INTERFACE I_XP_Environment  EXTENDS __SYSTEM.IQueryInterface, I_CH_Object

METHOD AddToGroup : HRESULT
VAR_INPUT
	iGroup : I_XP_Group;
END_VAR
END_METHOD

METHOD Clear : HRESULT
END_METHOD

METHOD Configure : HRESULT
VAR_INPUT
END_VAR
END_METHOD

{attribute 'monitoring':='call'}
PROPERTY Feedback : I_XP_Feedback
GET
END_GET
END_PROPERTY

METHOD Initialize : HRESULT
END_METHOD

{attribute 'monitoring':='call'}
PROPERTY Mapped : BOOL //Project is mapped to MC (McToPlc and PlcToMc)
GET
END_GET
END_PROPERTY

{attribute 'monitoring':='call'}
//Unique object ID
PROPERTY OID : OTCID
GET
END_GET
END_PROPERTY

{attribute 'monitoring':='call'}
PROPERTY PlanarEnvironment : REFERENCE TO MC_PlanarEnvironment
GET
END_GET
END_PROPERTY

METHOD RemoveFromGroup : HRESULT
END_METHOD

METHOD PUBLIC Update : HRESULT
VAR_INPUT
END_VAR
END_METHOD

{attribute 'monitoring':='call'}
PROPERTY UtilityEnvirement : Tc3_XPlanarUtility.I_Environment
GET
END_GET
END_PROPERTY

END_INTERFACE

(* stored: Version 1.1.0.1, ProductVersion 3.1.4024.12
   Itf I_XP_Environment: Id {82d4e6a8-d939-49b0-818e-86b258207442}
   Method AddToGroup: Id {f4493e59-ad90-4dac-89cb-3c35b7abff5c}
   Method Clear: Id {2eaf657c-b06a-4ac5-8bfd-2f4b4ad6572c}
   Method Configure: Id {9bbca1e7-a2f1-485d-8de7-8f90a1dc3677}
   Property Feedback: Id {e6ee7906-45bb-443c-afb3-2b2a9b508770}
   Get Get: Id {cc18bd10-41f4-4051-8a16-631b92b39a61}
   Method Initialize: Id {0d86c81e-3fa8-49c7-87ef-1a4588a06d1e}
   Property Mapped: Id {14b61345-b383-42ca-9c63-97777c6507b6}
   Get Get: Id {def7e364-4983-49a2-8c16-a97e170bf491}
   Property OID: Id {d57780a8-d816-4f3a-87e8-b26abdce176d}
   Get Get: Id {392b3d6c-8a64-48ae-8401-41ec1794064d}
   Property PlanarEnvironment: Id {d65c920f-3d4e-48f7-ae43-79864570d93f}
   Get Get: Id {23f8d9b1-51ed-469b-8515-26a29f4d1b5e}
   Method RemoveFromGroup: Id {0c2f8f63-9e17-4cfb-8064-d9613a987c2a}
   Method Update: Id {59e802b9-e7ee-42b2-909a-2e831ace6dc5}
   Property UtilityEnvirement: Id {fd24b682-4ff6-4ca5-a2e9-fb815df216ce}
   Get Get: Id {3f66a6a5-9ba4-4ba0-923f-e7c56dd321a6} *)
